ABB RobotStudio station: ExamProject.rspag

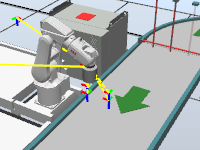
--- station ---
Station Station (saved by RobotStudio 20.4.9280.0)
Controller Controller
  mechanical unit ROB_1: IRB120_3_58__01, 6 joints, base frame (-2180.11, -2836.83, 440) mm, rotated rx 0 ry 0 rz 180 deg
  mechanical unit ROB_2: IRB120_3_58__01_2, 6 joints, base frame (-2037.23, -376.03, 440) mm, rotated rx 0 ry 0 rz 135 deg
Layout (positions relative to the parent item):
  - EksamensProjekt [graphiccomponentgroup]
    - Node3 [part] at (-2371.37, -6819.79, 495) mm
    - Node8 [part] at (-2371.37, -5982.29, 490) mm
    - Node11 [part] at (-2371.37, -5982.29, 475) mm, rotated rx 0 ry 0 rz -180 deg
    - Node12 [part] at (-2030.37, -6982.29, 230) mm, rotated rx 0 ry 0 rz -180 deg
    - Node13 [part] at (-2712.37, -6982.29, 230) mm, rotated rx 0 ry 0 rz -180 deg
    - Node14 [part] at (-2030.37, -6982.29, 15) mm, rotated rx 0 ry 0 rz -180 deg
    - Node15 [part] at (-2712.37, -6982.29, 15) mm, rotated rx 0 ry 0 rz -180 deg
    - Node16 [part] at (-2030.37, -4982.29, 230) mm, rotated rx 0 ry 0 rz -180 deg
    - Node17 [part] at (-2712.37, -4982.29, 230) mm, rotated rx 0 ry 0 rz -180 deg
    - Node18 [part] at (-2030.37, -4982.29, 15) mm, rotated rx 0 ry 0 rz -180 deg
    - Node19 [part] at (-2712.37, -4982.29, 15) mm, rotated rx 0 ry 0 rz -180 deg
    - Node20 [part] at (-2712.37, -5982.29, 475) mm, rotated rx 0 ry 90 rz -180 deg
    - Node21 [part] at (-2030.37, -5982.29, 475) mm, rotated rx 0 ry 90 rz -180 deg
    - Node28 [part] at (-2012.29, -1621.87, 440) mm
    - Node31 [part] at (-2012.29, -1621.87, 425) mm, rotated rx 0 ry 0 rz 180 deg
    - Node32 [part] at (-1671.29, -2621.87, 205) mm, rotated rx 0 ry 0 rz 180 deg
    - Node33 [part] at (-2353.29, -2621.87, 205) mm, rotated rx 0 ry 0 rz 180 deg
    - Node34 [part] at (-1671.29, -2621.87, 15) mm, rotated rx 0 ry 0 rz 180 deg
    - Node35 [part] at (-2353.29, -2621.87, 15) mm, rotated rx 0 ry 0 rz 180 deg
    - Node36 [part] at (-1671.29, -621.87, 205) mm, rotated rx 0 ry 0 rz 180 deg
    - Node37 [part] at (-2353.29, -621.87, 205) mm, rotated rx 0 ry 0 rz 180 deg
    - Node38 [part] at (-1671.29, -621.87, 15) mm, rotated rx 0 ry 0 rz 180 deg
    - Node39 [part] at (-2353.29, -621.87, 15) mm, rotated rx 0 ry 0 rz 180 deg
    - Node40 [part] at (-2353.29, -1621.87, 425) mm, rotated rx 0 ry 90 rz 180 deg
    - Node41 [part] at (-1671.29, -1621.87, 425) mm, rotated rx 0 ry 90 rz 180 deg
    - Node42 [part] at (-1000, -3057.54, 497) mm
    - Node43 [part] at (-1000, -3267.54, 497) mm, rotated rx 0 ry 0 rz -90 deg
    - Node44 [part] at (-1000, -3720.43, 497) mm, rotated rx 0 ry 0 rz 180 deg
    - Node45 [part] at (-1000, -3510.43, 497) mm, rotated rx 0 ry 0 rz 90 deg
    - Node46 [part] at (-4642.21, -2659.95, 161) mm
    - Node48 [part] at (-2388.44, -718.97, 510) mm, rotated rx 0 ry 0 rz 180 deg
    - Node49 [part] at (-1706.44, -718.97, 510) mm
    - Node51 [part] at (-2047.44, -718.97, 510) mm, rotated rx 0 ry 0 rz 180 deg
    - Node52 [part] at (-1000, -3200, 960) mm, rotated rx 90 ry 0 rz 0 deg
    - Node53 [part] at (-1000, -3200, 700) mm, rotated rx 174.29 ry 90 rz 84.29 deg
    - Node54 [part] at (-1000, -3550, 960) mm, rotated rx 90 ry 0 rz 0 deg
    - Node55 [part] at (-1000, -3550, 700) mm, rotated rx 174.29 ry 90 rz 84.29 deg
    - Node62 [part] at (-3419.43, -2666.76, 440) mm, rotated rx 0 ry 0 rz 90 deg
    - Node65 [part] at (-3419.44, -2666.76, 425) mm, rotated rx 0 ry 0 rz -90 deg
    - Node66 [part] at (-2419.43, -2325.76, 205) mm, rotated rx 0 ry 0 rz -90 deg
    - Node67 [part] at (-2419.44, -3007.76, 205) mm, rotated rx 0 ry 0 rz -90 deg
    - Node68 [part] at (-2419.43, -2325.76, 15) mm, rotated rx 0 ry 0 rz -90 deg
    - Node69 [part] at (-2419.44, -3007.76, 15) mm, rotated rx 0 ry 0 rz -90 deg
    - Node70 [part] at (-4419.44, -2325.76, 205) mm, rotated rx 0 ry 0 rz -90 deg
    - Node71 [part] at (-4419.44, -3007.76, 205) mm, rotated rx 0 ry 0 rz -90 deg
    - Node72 [part] at (-4419.44, -2325.76, 15) mm, rotated rx 0 ry 0 rz -90 deg
    - Node73 [part] at (-4419.44, -3007.76, 15) mm, rotated rx 0 ry 0 rz -90 deg
    - Node74 [part] at (-3419.44, -3007.76, 425) mm, rotated rx 0 ry 90 rz -90 deg
    - Node75 [part] at (-3419.43, -2325.76, 425) mm, rotated rx 0 ry 90 rz -90 deg
    - Node76 [part] at (-1000, -3375, 960) mm, rotated rx 90 ry 0 rz 0 deg
    - Node77 [part] at (-1000, -3375, 700) mm, rotated rx 174.29 ry 90 rz 84.29 deg
    - Node79 [part] at (-962.99, -2500.53, 99.06) mm
    - Node80 [part] at (-962.99, -2500.53, 99.06) mm
    - Node81 [part] at (-962.99, -2500.53, 99.06) mm
    - Node82 [part] at (-962.99, -2500.53, 99.06) mm
    - Node83 [part] at (-962.99, -2500.53, 99.06) mm
    - Node84 [part] at (-962.99, -2500.53, 99.06) mm
    - Node85 [part] at (-962.99, -2500.53, 99.06) mm
    - Node86 [part] at (-1080.86, -2495.4, 636.21) mm
    - Node95 [part] at (-2163.95, -2817.97, 425) mm, rotated rx 0 ry 0 rz -1.03 deg
    - Node96 [part] at (-2351.77, -2639.57, 205) mm, rotated rx 0 ry 0 rz -1.03 deg
    - Node97 [part] at (-1969.83, -2646.44, 205) mm, rotated rx 0 ry 0 rz -1.03 deg
    - Node98 [part] at (-2351.77, -2639.57, 15) mm, rotated rx 0 ry 0 rz -1.03 deg
    - Node99 [part] at (-1969.83, -2646.44, 15) mm, rotated rx 0 ry 0 rz -1.03 deg
    - Node100 [part] at (-2358.07, -2989.51, 205) mm, rotated rx 0 ry 0 rz -1.03 deg
    - Node101 [part] at (-1976.13, -2996.38, 205) mm, rotated rx 0 ry 0 rz -1.03 deg
    - Node102 [part] at (-2358.07, -2989.51, 15) mm, rotated rx 0 ry 0 rz -1.03 deg
    - Node103 [part] at (-1976.13, -2996.38, 15) mm, rotated rx 0 ry 0 rz -1.03 deg
    - Node104 [part] at (-1972.98, -2821.41, 425) mm, rotated rx -85.62 ry 90 rz -86.65 deg
    - Node105 [part] at (-2354.92, -2814.54, 425) mm, rotated rx -85.62 ry 90 rz -86.65 deg
    - Node114 [part] at (-2048.93, -380.61, 425) mm, rotated rx 0 ry 0 rz -1.03 deg
    - Node115 [part] at (-2236.75, -202.2, 205) mm, rotated rx 0 ry 0 rz -1.03 deg
    - Node116 [part] at (-1854.81, -209.07, 205) mm, rotated rx 0 ry 0 rz -1.03 deg
    - Node117 [part] at (-2236.75, -202.2, 15) mm, rotated rx 0 ry 0 rz -1.03 deg
    - Node118 [part] at (-1854.81, -209.07, 15) mm, rotated rx 0 ry 0 rz -1.03 deg
    - Node119 [part] at (-2243.04, -552.14, 205) mm, rotated rx 0 ry 0 rz -1.03 deg
    - Node120 [part] at (-1861.1, -559.01, 205) mm, rotated rx 0 ry 0 rz -1.03 deg
    - Node121 [part] at (-2243.04, -552.14, 15) mm, rotated rx 0 ry 0 rz -1.03 deg
    - Node122 [part] at (-1861.1, -559.01, 15) mm, rotated rx 0 ry 0 rz -1.03 deg
    - Node123 [part] at (-1857.96, -384.04, 425) mm, rotated rx -85.62 ry 90 rz -86.65 deg
    - Node124 [part] at (-2239.9, -377.17, 425) mm, rotated rx -85.62 ry 90 rz -86.65 deg
    - Node132 [part] at (-2180.11, -2836.83, 440) mm, rotated rx 78.69 ry -90 rz 9.51 deg
    - Node188 [part] at (-1384.63, 119.54, 0) mm, rotated rx 0 ry 90 rz 90 deg
    - Node189 [part] at (-1384.63, 119.54, 0) mm, rotated rx 0 ry 90 rz 90 deg
    - Node191 [part] at (-2010.83, 559.9, 0) mm, rotated rx 0 ry 90 rz -90 deg
    - Node192 [part] at (-2010.83, 559.9, 0) mm, rotated rx 0 ry 90 rz -90 deg
    - Node193 [part] at (-2010.83, 559.9, 0) mm, rotated rx 0 ry 90 rz -90 deg
    - Node196 [part] at (-2642.02, 96.05, 0) mm, rotated rx 0 ry 90 rz 90 deg
    - Node197 [part] at (-2642.02, 96.05, 0) mm, rotated rx 0 ry 90 rz 90 deg
    - Node207 [part] at (-872.91, -4039.09, 425) mm, rotated rx 0 ry 0 rz -180 deg
    - Node208 [part] at (-413.29, -3579.47, 440) mm, rotated rx 0 ry 0 rz 45 deg
    - Node217 [part] at (-872.91, -4039.09, 425) mm, rotated rx 0 ry 0 rz -180 deg
    - Node218 [part] at (-872.91, -4039.09, 425) mm, rotated rx 0 ry 0 rz -180 deg
    - Node225 [part] at (-1872.91, -4689.09, 440) mm, rotated rx 0 ry 0 rz -90 deg
    - Node228 [part] at (-1872.91, -4689.09, 425) mm, rotated rx 0 ry 0 rz 90 deg
    - Node229 [part] at (-2872.91, -5030.09, 205) mm, rotated rx 0 ry 0 rz 90 deg
    - Node230 [part] at (-2872.91, -4348.09, 205) mm, rotated rx 0 ry 0 rz 90 deg
    - Node231 [part] at (-2872.91, -5030.09, 15) mm, rotated rx 0 ry 0 rz 90 deg
    - Node232 [part] at (-2872.91, -4348.09, 15) mm, rotated rx 0 ry 0 rz 90 deg
    - Node233 [part] at (-872.91, -5030.09, 205) mm, rotated rx 0 ry 0 rz 90 deg
    - Node234 [part] at (-872.91, -4348.09, 205) mm, rotated rx 0 ry 0 rz 90 deg
    - Node235 [part] at (-872.91, -5030.09, 15) mm, rotated rx 0 ry 0 rz 90 deg
    - Node236 [part] at (-872.91, -4348.09, 15) mm, rotated rx 0 ry 0 rz 90 deg
    - Node237 [part] at (-1872.91, -4348.09, 425) mm, rotated rx 0 ry 90 rz 90 deg
    - Node238 [part] at (-1872.91, -5030.09, 402.5) mm, rotated rx 0 ry 90 rz 90 deg
    - Node248 [part] at (-872.91, -4039.09, 425) mm, rotated rx 0 ry 0 rz 90 deg
    - Node249 [part] at (-413.29, -4498.71, 440) mm, rotated rx 0 ry 0 rz -45 deg
    - Node258 [part] at (-872.91, -4039.09, 425) mm, rotated rx 0 ry 0 rz 90 deg
    - Node259 [part] at (-872.91, -4039.09, 425) mm, rotated rx 0 ry 0 rz 90 deg
    - Node269 [part] at (-2872.91, -4039.09, 425) mm, rotated rx 0 ry 0 rz -90 deg
    - Node270 [part] at (-3332.53, -3579.47, 440) mm, rotated rx 0 ry 0 rz 135 deg
    - Node279 [part] at (-2872.91, -4039.09, 425) mm, rotated rx 0 ry 0 rz -90 deg
    - Node280 [part] at (-2872.91, -4039.09, 425) mm, rotated rx 0 ry 0 rz -90 deg
    - Node290 [part] at (-2872.91, -4039.09, 425) mm
    - Node291 [part] at (-3332.53, -4498.71, 440) mm, rotated rx 0 ry 0 rz -135 deg
    - Node300 [part] at (-2872.91, -4039.09, 425) mm
    - Node301 [part] at (-2872.91, -4039.09, 425) mm
    - Node308 [part] at (-1872.91, -3389.09, 440) mm, rotated rx 0 ry 0 rz 90 deg
    - Node311 [part] at (-1872.91, -3389.09, 425) mm, rotated rx 0 ry 0 rz -90 deg
    - Node312 [part] at (-872.91, -3048.09, 205) mm, rotated rx 0 ry 0 rz -90 deg
    - Node313 [part] at (-872.91, -3730.09, 205) mm, rotated rx 0 ry 0 rz -90 deg
    - Node314 [part] at (-872.91, -3048.09, 15) mm, rotated rx 0 ry 0 rz -90 deg
    - Node315 [part] at (-872.91, -3730.09, 15) mm, rotated rx 0 ry 0 rz -90 deg
    - Node316 [part] at (-2872.91, -3048.09, 205) mm, rotated rx 0 ry 0 rz -90 deg
    - Node317 [part] at (-2872.91, -3730.09, 205) mm, rotated rx 0 ry 0 rz -90 deg
    - Node318 [part] at (-2872.91, -3048.09, 15) mm, rotated rx 0 ry 0 rz -90 deg
    - Node319 [part] at (-2872.91, -3730.09, 15) mm, rotated rx 0 ry 0 rz -90 deg
    - Node320 [part] at (-1872.91, -3730.09, 425) mm, rotated rx 0 ry 90 rz -90 deg
    - Node321 [part] at (-1872.91, -3048.09, 425) mm, rotated rx 0 ry 90 rz -90 deg
    - Node533 [part] at (-2037.23, -376.03, 440) mm, rotated rx 78.69 ry -90 rz -31.89 deg
    - Node794 [part] at (-1527.67, -303.76, 425) mm
    - Node795 [part] at (-2062.04, -30.96, 425) mm
    - Node796 [part] at (-2436.77, -305.66, 425) mm
  - IRB120_3_58__01 [mechanism, from Robots\IRB120_3_58_G_01.rslib] at (-2180.11, -2836.83, 440) mm, rotated rx 0 ry 0 rz 180 deg; joint values [1.5712, 0.2361, 0.2235, 0.0005, 1.1183, -0.0001] (rad or m)
  - IRB120_3_58__01_2 [mechanism, from Robots\IRB120_3_58_G_01.rslib] at (-2037.23, -376.03, 440) mm, rotated rx 0 ry 0 rz 135 deg; joint values [2.3486, 0.5389, -0.5356, -0.0097, 1.5677, -0.002] (rad or m)
  - SimpleGripperTool [mechanism] at (-2179.91, -3201.18, 849.29) mm, rotated rx 179.97 ry -0.41 rz 90.02 deg
      TCP SimpleGripperTool at (0, 0, 0) mm
      links: SimpleGripper
  - SimpleGripperTool [mechanism] at (-2041.29, -816.79, 958.73) mm, rotated rx -179.45 ry -0.01 rz 89.68 deg
      TCP SimpleGripperTool at (0, 0, 0) mm
      links: SimpleGripper_2
Attachment: SimpleGripperTool is attached to IRB120_3_58__01 / Link6
Attachment: SimpleGripperTool is attached to IRB120_3_58__01_2 / Link6
Targets, tools, work objects and paths stored in the station and not in the controller backup, written as RAPID:
! task T_ROB2
MODULE Module1
  PROC Path_Pickup_L_Home()
    MoveJ Target2_Pickup_S,v1000,z100,tool0\WObj:=wobj0;
    MoveJ Target2_Home,v1000,z100,tool0\WObj:=wobj0;
  ENDPROC
  PROC Path_Pickup_S_Home()
    MoveJ Target2_Pickup_L,v1000,z100,tool0\WObj:=wobj0;
    MoveJ Target2_Home,v1000,z100,tool0\WObj:=wobj0;
  ENDPROC
ENDMODULE


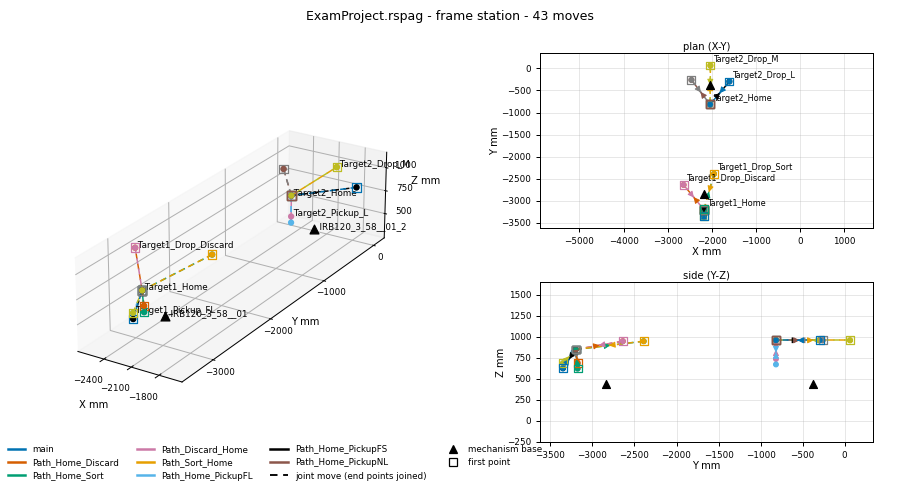
[picture p0: tool path of ExamProject.rspag in frame station, 43 of 43 moves have a stored position in this frame; points joined in program order, loops and branches not executed]
--- Backups/Controller/RAPID/TASK1/PROGMOD/CalibData.mod ---
MODULE CalibData
    PERS tooldata SimpleGripperTool:=[TRUE,[[0,0,0],[1,0,0,0]],[1,[0,0,1],[1,0,0,0],0,0,0]];
ENDMODULE

--- Backups/Controller/RAPID/TASK1/PROGMOD/Module1.mod ---
MODULE Module1
        CONST robtarget Target1_Home:=[[-2179.911939957,-3201.183818015,849.285443701],[0.002346881,-0.707006801,-0.707197774,-0.002680418],[1,0,-1,0],[9E+09,9E+09,9E+09,9E+09,9E+09,9E+09]];
    CONST robtarget Target1_Pickup_FL:=[[-2179.911934246,-3351.083079924,685.839453438],[0.002346893,-0.70700679,-0.707197785,-0.00268043],[1,0,-1,0],[9E+09,9E+09,9E+09,9E+09,9E+09,9E+09]];
    CONST robtarget Target1_Pickup_FS:=[[-2179.911934232,-3351.083078073,625.182449341],[0.002346896,-0.707006801,-0.707197774,-0.002680433],[1,0,-1,0],[9E+09,9E+09,9E+09,9E+09,9E+09,9E+09]];
    CONST robtarget Target1_Pickup_NL:=[[-2179.911950334,-3176.803980267,685.839457445],[0.002346877,-0.707006801,-0.707197774,-0.002680414],[1,0,-1,0],[9E+09,9E+09,9E+09,9E+09,9E+09,9E+09]];
    CONST robtarget Target1_Pickup_NS:=[[-2179.911950358,-3176.803984153,622.544451269],[0.002346864,-0.707006801,-0.707197774,-0.002680401],[1,0,-1,0],[9E+09,9E+09,9E+09,9E+09,9E+09,9E+09]];
    CONST robtarget Target1_Drop_Discard:=[[-2640.444699172,-2638.477494089,947.558490472],[0.000236373,0.999993654,-0.00001496,0.003554735],[-1,-1,-1,0],[9E+09,9E+09,9E+09,9E+09,9E+09,9E+09]];
    CONST robtarget Target1_Drop_Sort:=[[-1951.858716039,-2390.564268364,947.558490472],[0.002756603,0.683400301,-0.730035161,0.002256802],[-2,-1,-1,0],[9E+09,9E+09,9E+09,9E+09,9E+09,9E+09]];
!***********************************************************
    !
    ! Module:  Module1
    !
    ! Description:
    !   <Insert description here>
    !
    ! Author: mathi
    !
    ! Version: 1.0
    !
    !***********************************************************


    !***********************************************************
    !
    ! Procedure main
    !
    !   This is the entry point of your program
    !
    !***********************************************************
    PROC main()
        IF DInput(diInitHome1) = 1 THEN
            MoveJ Target1_Home,v1000,z100,SimpleGripperTool\WObj:=wobj0;

        ELSEIF DInput(diPickFL1) = 1 THEN
            IF DInput(diHome1) = 0 THEN
                SetDO doInPosition1,0;
                Path_Home_PickupFL;
                SetDO doInPosition1,1;
            ELSE
                SetDO doInPosition1, 0;
                Path_PickupFL_Home;
                SetDO doInPosition1, 1;
            ENDIF

        ELSEIF DInput(diPickFS1) = 1 THEN
            IF DInput(diHome1) = 0 THEN
                SetDO doInPosition1,0;
                Path_Home_PickupFS;
                SetDO doInPosition1,1;
            ELSE
                SetDO doInPosition1, 0;
                Path_PickupFS_Home;
                SetDO doInPosition1, 1;
            ENDIF

        ELSEIF DInput(diPickNL1) = 1 THEN
            IF DInput(diHome1) = 0 THEN
                SetDO doInPosition1,0;
                Path_Home_PickupNL;
                SetDO doInPosition1,1;
            ELSE
                SetDO doInPosition1, 0;
                Path_PickupNL_Home;
                SetDO doInPosition1, 1;
            ENDIF

        ELSEIF DInput(diHomeDiscard1) = 1 THEN
            IF DInput(diHome1) = 0 THEN
                SetDO doInPosition1,0;
                Path_Home_Discard;
                SetDO doInPosition1,1;
            ELSE
                SetDO doInPosition1, 0;
                Path_Discard_Home;
                SetDO doInPosition1, 1;
            ENDIF

        ELSEIF DInput(diHomeSort1) = 1 THEN
            IF DInput(diHome1) = 0 THEN
                SetDO doInPosition1,0;
                Path_Home_Sort;
                SetDO doInPosition1,1;
            ELSE
                SetDO doInPosition1, 0;
                Path_Sort_Home;
                SetDO doInPosition1, 1;
            ENDIF

        ELSEIF DInput(diPickFL1) = 1 THEN
            IF DInput(diHome1) = 0 THEN
                SetDO doInPosition1,0;
                Path_Home_PickupFL;
                SetDO doInPosition1,1;
            ELSE
                SetDO doInPosition1, 0;
                Path_PickupFL_Home;
                SetDO doInPosition1, 1;
            ENDIF
        ENDIF


    ENDPROC
    PROC Path_Home_Discard()
        MoveJ Target1_Home,v1000,z100,SimpleGripperTool\WObj:=wobj0;
        MoveJ Target1_Drop_Discard,v1000,z100,SimpleGripperTool\WObj:=wobj0;
    ENDPROC
    PROC Path_Home_Sort()
        MoveJ Target1_Home,v1000,z100,SimpleGripperTool\WObj:=wobj0;
        MoveJ Target1_Drop_Sort,v1000,z100,SimpleGripperTool\WObj:=wobj0;
    ENDPROC
    PROC Path_Discard_Home()
        MoveJ Target1_Drop_Discard,v1000,z100,SimpleGripperTool\WObj:=wobj0;
        MoveJ Target1_Home,v1000,z100,SimpleGripperTool\WObj:=wobj0;
    ENDPROC
    PROC Path_Sort_Home()
        MoveJ Target1_Drop_Sort,v1000,z100,SimpleGripperTool\WObj:=wobj0;
        MoveJ Target1_Home,v1000,z100,SimpleGripperTool\WObj:=wobj0;
    ENDPROC
    PROC Path_Home_PickupFL()
        MoveJ Target1_Home,v1000,z100,SimpleGripperTool\WObj:=wobj0;
        MoveJ Target1_Pickup_FL,v1000,z100,SimpleGripperTool\WObj:=wobj0;
    ENDPROC
    PROC Path_Home_PickupFS()
        MoveJ Target1_Home,v1000,z100,SimpleGripperTool\WObj:=wobj0;
        MoveJ Target1_Pickup_FS,v1000,z100,SimpleGripperTool\WObj:=wobj0;
    ENDPROC
    PROC Path_Home_PickupNL()
        MoveJ Target1_Home,v1000,z100,SimpleGripperTool\WObj:=wobj0;
        MoveJ Target1_Pickup_NL,v1000,z100,SimpleGripperTool\WObj:=wobj0;
    ENDPROC
    PROC Path_Home_PickupNS()
        MoveJ Target1_Home,v1000,z100,SimpleGripperTool\WObj:=wobj0;
        MoveJ Target1_Pickup_NS,v1000,z100,SimpleGripperTool\WObj:=wobj0;
    ENDPROC
    PROC Path_PickupFL_Home()
        MoveJ Target1_Pickup_FL,v1000,z100,SimpleGripperTool\WObj:=wobj0;
        MoveJ Target1_Home,v1000,z100,SimpleGripperTool\WObj:=wobj0;
    ENDPROC
    PROC Path_PickupFS_Home()
        MoveJ Target1_Pickup_FS,v1000,z100,SimpleGripperTool\WObj:=wobj0;
        MoveJ Target1_Home,v1000,z100,SimpleGripperTool\WObj:=wobj0;
    ENDPROC
    PROC Path_PickupNL_Home()
        MoveJ Target1_Pickup_NL,v1000,z100,SimpleGripperTool\WObj:=wobj0;
        MoveJ Target1_Home,v1000,z100,SimpleGripperTool\WObj:=wobj0;
    ENDPROC
    PROC Path_PickupNS_Home()
        MoveJ Target1_Pickup_NS,v1000,z100,SimpleGripperTool\WObj:=wobj0;
        MoveJ Target1_Home,v1000,z100,SimpleGripperTool\WObj:=wobj0;
    ENDPROC
ENDMODULE

--- Backups/Controller/RAPID/TASK2/PROGMOD/Module1.mod ---
MODULE Module1
        CONST robtarget Target2_Home:=[[-2041.291356005,-816.791303667,958.7300671],[0.003500372,-0.709065794,-0.705125793,0.00332614],[1,-1,-1,0],[9E+09,9E+09,9E+09,9E+09,9E+09,9E+09]];
    CONST robtarget Target2_Pickup_L:=[[-2041.291355914,-816.791293008,736.319944451],[0.003500375,-0.709065794,-0.705125793,0.003326137],[1,-1,0,0],[9E+09,9E+09,9E+09,9E+09,9E+09,9E+09]];
    CONST robtarget Target2_Drop_M:=[[-2033.790669408,64.736596316,958.7300671],[0.003328609,-0.705625949,0.708568066,-0.003498024],[-1,-1,-1,0],[9E+09,9E+09,9E+09,9E+09,9E+09,9E+09]];
    CONST robtarget Target2_Pickup_S:=[[-2041.291355787,-816.791291264,670.969863629],[0.003500367,-0.709065794,-0.705125793,0.003326144],[1,-1,0,0],[9E+09,9E+09,9E+09,9E+09,9E+09,9E+09]];
    CONST robtarget Target2_Drop_L:=[[-1603.663890462,-296.610543419,958.7300671],[0.00033616,-0.092272904,0.995722047,-0.004816929],[-2,-1,-1,0],[9E+09,9E+09,9E+09,9E+09,9E+09,9E+09]];
    CONST robtarget Target2_Drop_S:=[[-2462.839523363,-261.384655368,958.7300671],[0.004772627,-0.991584,0.129374864,-0.00073338],[0,-1,-1,0],[9E+09,9E+09,9E+09,9E+09,9E+09,9E+09]];
!***********************************************************
    !
    ! Module:  Module1
    !
    ! Description:
    !   <Insert description here>
    !
    ! Author: mathi
    !
    ! Version: 1.0
    !
    !***********************************************************


    !***********************************************************
    !
    ! Procedure main
    !
    !   This is the entry point of your program
    !
    !***********************************************************
    PROC main()
        !Add your code here
    ENDPROC
    PROC Path_Pickup_L()
        MoveJ Target2_Home,v1000,z100,tool0\WObj:=wobj0;
        MoveJ Target2_Pickup_L,v1000,z100,tool0\WObj:=wobj0;
        MoveJ Target2_Home,v1000,z100,tool0\WObj:=wobj0;
    ENDPROC
    PROC Path_Drop_M()
        MoveJ Target2_Home,v1000,z100,tool0\WObj:=wobj0;
        MoveJ Target2_Drop_M,v1000,z100,tool0\WObj:=wobj0;
    ENDPROC
    PROC Path_Pickup_S()
        MoveJ Target2_Home,v1000,z100,tool0\WObj:=wobj0;
        MoveJ Target2_Pickup_S,v1000,z100,tool0\WObj:=wobj0;
        MoveJ Target2_Home,v1000,z100,tool0\WObj:=wobj0;
    ENDPROC
    PROC Path_Drop_L()
        MoveJ Target2_Home,v1000,z100,tool0\WObj:=wobj0;
        MoveJ Target2_Drop_L,v1000,z100,tool0\WObj:=wobj0;
    ENDPROC
    PROC Path_Drop_S()
        MoveJ Target2_Home,v1000,z100,tool0\WObj:=wobj0;
        MoveJ Target2_Drop_S,v1000,z100,tool0\WObj:=wobj0;
    ENDPROC
    PROC Path_S_Home()
        MoveJ Target2_Drop_S,v1000,z100,tool0\WObj:=wobj0;
        MoveJ Target2_Home,v1000,z100,tool0\WObj:=wobj0;
    ENDPROC
    PROC Path_M_Home()
        MoveJ Target2_Drop_M,v1000,z100,tool0\WObj:=wobj0;
        MoveJ Target2_Home,v1000,z100,tool0\WObj:=wobj0;
    ENDPROC
    PROC Path_L_Home()
        MoveJ Target2_Drop_L,v1000,z100,tool0\WObj:=wobj0;
        MoveJ Target2_Home,v1000,z100,tool0\WObj:=wobj0;
    ENDPROC
ENDMODULE

--- Backups/Controller/SYSPAR/EIO.cfg ---
EIO:CFG_1.0:6:1::
#
EIO_SIGNAL:

      -Name "doGrip1" -SignalType "DO" -Category "Gripper" -Access "All"

      -Name "doGrip2" -SignalType "DO" -Category "Gripper" -Access "All"

      -Name "diPickNS1" -SignalType "DI" -Category "Robot1" -Access "All"

      -Name "diPickNL1" -SignalType "DI" -Category "Robot1" -Access "All"

      -Name "diPickFL1" -SignalType "DI" -Category "Robot1" -Access "All"

      -Name "diPickFS1" -SignalType "DI" -Category "Robot1" -Access "All"

      -Name "diHomeDiscard1" -SignalType "DI" -Category "Robot1" -Access "All"

      -Name "diDiscardHome1" -SignalType "DI" -Category "Robot1" -Access "All"

      -Name "diHomeSort1" -SignalType "DI" -Category "Robot1" -Access "All"

      -Name "diSortHome1" -SignalType "DI" -Category "Robot1" -Access "All"

      -Name "diPickS2" -SignalType "DI" -Category "Robot2" -Access "All"

      -Name "diPickL2" -SignalType "DI" -Category "Robot2" -Access "All"

      -Name "diHomeS2" -SignalType "DI" -Category "Robot2" -Access "All"

      -Name "diHomeM2" -SignalType "DI" -Category "Robot2" -Access "All"

      -Name "diHomeL2" -SignalType "DI" -Category "Robot2" -Access "All"

      -Name "doInPosition1" -SignalType "DO" -Category "robot1" -Access "All"

      -Name "doInPosition2" -SignalType "DO" -Category "Robot2" -Access "All"

      -Name "diHome1" -SignalType "DI" -Category "Robot1" -Access "All"

      -Name "diHome2" -SignalType "DI" -Category "Robot2" -Access "All"

      -Name "diInitHome1" -SignalType "DI" -Category "Robot1" -Access "All"

      -Name "diInitHome2" -SignalType "DI" -Category "Robot2" -Access "All"

      -Name "diPickM2" -SignalType "DI" -Category "Robot2" -Access "All"
